PROGRAM Cascading
VAR
END_VAR

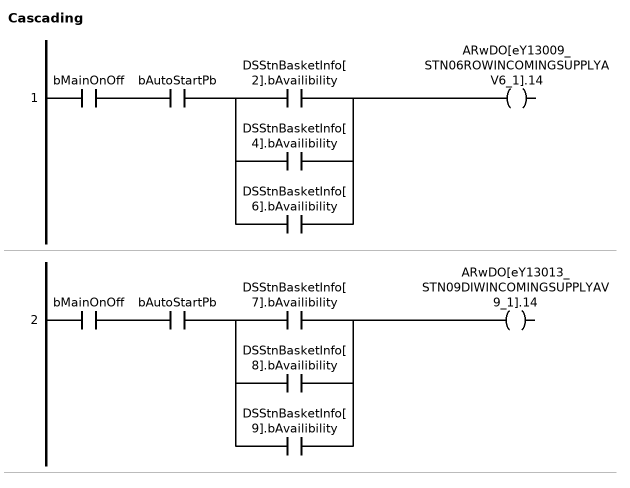
// NETWORK 1
ARwDO[eY13009_STN06ROWINCOMINGSUPPLYAV6_1].14 := bMainOnOff AND bAutoStartPb AND (DSStnBasketInfo[2].bAvailibility OR DSStnBasketInfo[4].bAvailibility OR DSStnBasketInfo[6].bAvailibility);

// NETWORK 2
ARwDO[eY13013_STN09DIWINCOMINGSUPPLYAV9_1].14 := bMainOnOff AND bAutoStartPb AND (DSStnBasketInfo[7].bAvailibility OR DSStnBasketInfo[8].bAvailibility OR DSStnBasketInfo[9].bAvailibility);

END_PROGRAM

(* stored: Version 1.1.0.1, ProductVersion 3.1.4024.12
   POU Cascading: Id {7bfa9efd-dad7-4dc2-8e34-4754c88b302c}, SpecialFunc None *)
